// TIA Portal V17 export
// export: Created 2026-04-13T11:12:42.4666713Z, ExportSetting WithDefaults, DisplayName Totally Integrated Automation Portal, DisplayVersion V17 Update 4, DisplayName TIA Portal Openness, DisplayVersion V17 Update 4, DisplayName TIA Portal Version Control Interface, DisplayVersion V17, DisplayName SINAMICS Startdrive Advanced, DisplayVersion V17, DisplayName SINAMICS Startdrive G130, G150, S120, S150, SINAMICS MV, S210, DisplayVersion V17, DisplayName SINAMICS Startdrive G110M, G120, G120C, G120D, G120P, G115D, DisplayVersion V17, DisplayName STEP 7 Professional, DisplayVersion V17 Update 4, DisplayName STEP 7 Safety, DisplayVersion V17, DisplayName WinCC Professional, DisplayVersion V17 Update 4
FUNCTION_BLOCK "0-模拟量滤波"   // FB109, LAD
{ S7_Optimized_Access := 'TRUE' }
VERSION : 0.1
// stored: AutoNumber true, IsIECCheckEnabled false, IsRetainMemResEnabled false, MemoryReserve 100, SetENOAutomatically false, UDAEnableTagReadback false
   VAR_INPUT
      模拟量数据输入 : Int;
      "上限(工程量)" : Real;
      "下限(工程量)" : Real := 100.0;
      "采样时间间隔（秒）" : Real := 1.0;
      滤波强度 : Int := 10;
   END_VAR
   VAR_OUTPUT
      工程量数据输出 : Real;
      "工程量数据输出(滤波后)" : Real;
      Error_MAX : Bool;
      Error_MIN : Bool;
   END_VAR
   VAR
      AI : Int;
      "Time" : Time;
      T0 { S7_SetPoint := 'True'} : TON_TIME;
      T1 { S7_SetPoint := 'True'} : TON_TIME;
      P0 { S7_SetPoint := 'True'} : R_TRIG;
      LB { S7_SetPoint := 'True'} : Array[1..20] of Real;
      ZS : Real;
      N : Int;
      stat滤波强度 : Int;
   END_VAR
BEGIN

REGION Network 1 (SCL)
   #Time:=DINT_TO_TIME( REAL_TO_DINT( #"采样时间间隔（秒）"*1000.0)-10);
   #T0(IN:=NOT #T1.Q,
       PT:=#Time);
   #T1(IN:=#T0.Q,
       PT:=T#10MS);
   #P0(CLK:=#T0.Q);



   #AI := #模拟量数据输入;
   IF #AI<0 THEN
       #AI := 0;
       #Error_MIN := 1;
   ELSE
       #Error_MIN := 0;
       ;
   END_IF;

   IF #AI>27648 THEN
       #AI := 27648;
       #Error_MAX := 1;
   ELSE
       #Error_MAX := 0;
       ;
   END_IF;
   #stat滤波强度 := #滤波强度;
   IF #滤波强度 > 20 THEN
       #stat滤波强度 := 20;
   END_IF;
   IF #滤波强度 < 1 THEN
       #stat滤波强度 := 1;
   END_IF;

   IF #P0.Q THEN
       #工程量数据输出 := INT_TO_REAL(#AI) / 27648.0 * (#"上限(工程量)" - #"下限(工程量)") + #"下限(工程量)";
       FOR #N := #stat滤波强度 TO 2 BY -1 DO
           #LB[#N] := #LB[#N - 1];
           ;
       END_FOR;
       #LB[1] := #工程量数据输出;

       #ZS := 0;
       FOR #N := 1 TO #stat滤波强度 DO
           #ZS := #ZS + #LB[#N];
       END_FOR;


       #"工程量数据输出(滤波后)" := #ZS / #stat滤波强度;



   END_IF;
END_REGION
END_FUNCTION_BLOCK
